{attribute 'qualified_only'}
{attribute 'strict'}
TYPE
E_Axis :
(
	X	:= 1,
	Y	:= 2,
	Z	:= 3
);
END_TYPE

(* stored: Version 1.1.0.1, ProductVersion 3.1.4024.12
   DUT E_Axis: Id {101823f3-54e0-47a0-8877-6216ee5bd2f1} *)
